(* PLC project Unnamed, Unknown Unnamed 1 *)
(* stored: creationDateTime 2021-10-04T15:01:11, modificationDateTime 2021-10-04T20:41:19 *)

PROGRAM part5a
  VAR
    MinLvlSensor AT %IX0.0 : BOOL;
    LowLvlSensor AT %IX0.1 : BOOL;
    MedLvlSensor AT %IX0.2 : BOOL;
    HighLvlSensor AT %IX0.3 : BOOL;
    InValve1_A AT %QX0.0 : BOOL;
    InValve2_B AT %QX0.1 : BOOL;
    InValve3_C AT %QX0.2 : BOOL;
    Blade AT %QX0.3 : BOOL;
    OutValve AT %QX0.4 : BOOL;
  END_VAR
  VAR
    State0 : BOOL := True;
    State1 : BOOL;
    State2 : BOOL;
    State3 : BOOL;
    State4 : BOOL;
    State5 : BOOL;
    State6 : BOOL;
    SR0 : SR;
    SR1 : SR;
    SR2 : SR;
    SR3 : SR;
    TON0 : TON;
    SR4 : SR;
    SR5 : SR;
    SR6 : SR;
    TON1 : TON;
  END_VAR

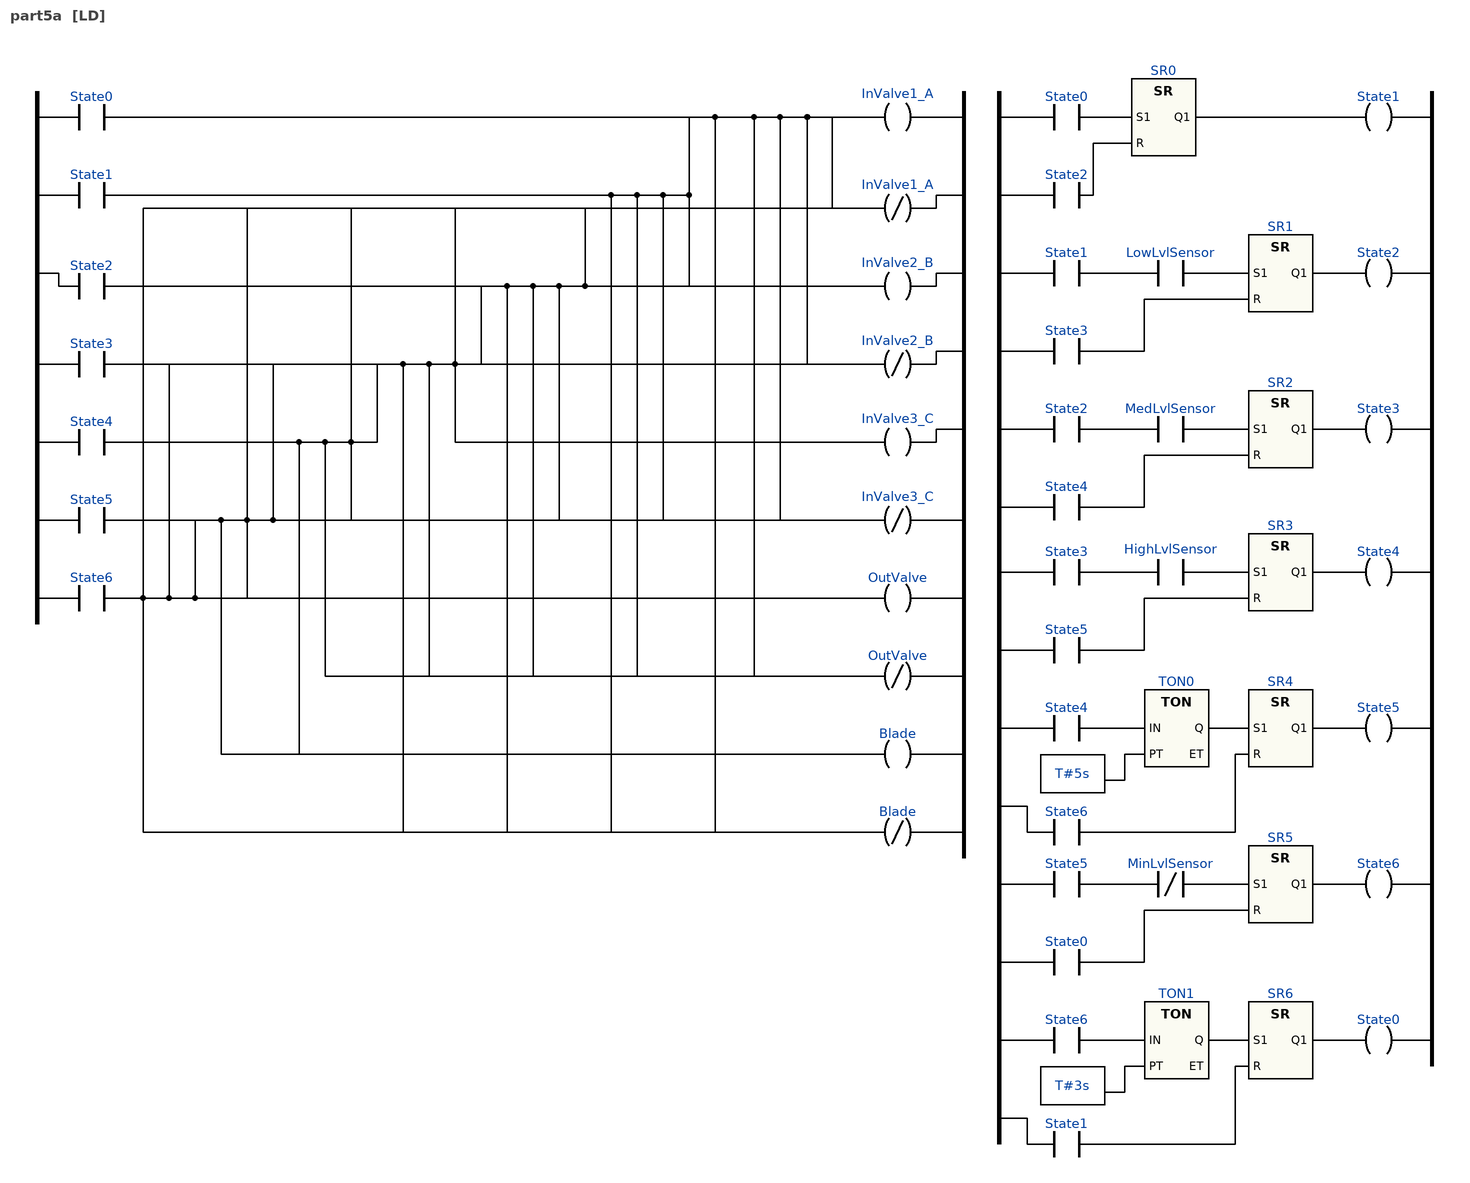
(* LD diagram, written out as Structured Text *)
InValve1_A := State1;
SR0(S1 := State0, R := State2);
State1 := SR0.Q1;
InValve1_A := NOT (State0 OR State2 OR State3 OR State4 OR State5 OR State6);
SR1(S1 := State1 AND LowLvlSensor, R := State3);
State2 := SR1.Q1;
InValve2_B := State1 OR State2 OR State3;
InValve2_B := NOT (State0 OR State4 OR State5 OR State6);
SR2(S1 := State2 AND MedLvlSensor, R := State4);
State3 := SR2.Q1;
InValve3_C := State3;
InValve3_C := NOT (State0 OR State1 OR State2 OR State4 OR State5 OR State6);
SR3(S1 := State3 AND HighLvlSensor, R := State5);
State4 := SR3.Q1;
OutValve := State5 OR State6;
OutValve := NOT (State0 OR State1 OR State2 OR State3 OR State4);
TON0(IN := State4, PT := T#5s);
SR4(S1 := TON0.Q, R := State6);
State5 := SR4.Q1;
Blade := State4 OR State5;
Blade := NOT (State0 OR State1 OR State2 OR State3 OR State6);
SR5(S1 := State5 AND NOT MinLvlSensor, R := State0);
State6 := SR5.Q1;
TON1(IN := State6, PT := T#3s);
SR6(S1 := TON1.Q, R := State1);
State0 := SR6.Q1;
END_PROGRAM

CONFIGURATION Config0
  RESOURCE Res0 ON PLC
    TASK task0(INTERVAL := T#20ms, PRIORITY := 0);
    PROGRAM instance0 WITH task0 : part5a;
  END_RESOURCE
END_CONFIGURATION
